FUNCTION_BLOCK FLOOR2_AR (* AR/ADI-Adapter-Wrapper um OSCAT FLOOR2 - bruckt zwischen adapter und OSCAT, ohne dass eine der beiden Basisbibliotheken von der anderen abhaengt *)
  (* Standard: 61499-2; Description: Copyright (c) 2026 Meisterschulen am Ostbahnhof This program and the accompanying materials are made available under the terms of the Eclipse Public License 2.0 which is available at https://www.eclipse.org/legal/epl-2.0/ SPDX-License-Identifier: EPL-2.0 *)
  (* Version 1.0, 2026-09-17, Franz Höpfinger, Meisterschulen am Ostbahnhof, Initial implementation of FLOOR2_AR wrapper FB - E_D_FF_ANY_1 als Aenderungsfilter (EO/ADI_OUT.E1 nur bei tatsaechlicher Wertaenderung), analog CTRL_PI_AR/FT_DERIV_AR in diesem Projekt *)
  PACKAGE OSCAT_adapter::Mathematical;
  (* Documentation:
  FLOOR2_AR
   🇩🇪 Deutsch
   Adapter-Wrapper um OSCAT::Basic::POUs::Mathematical::FLOOR2 (groesste ganze Zahl <= X, DINT-Variante von FLOOR fuer Werte ausserhalb des INT-Bereichs).
   Reine Adapter-Grenze
    - AR_IN (Socket, AR): Eingangssignal (REAL)
   - ADI_OUT (Plug, ADI): Ergebnis (DINT)
    E_D_FF_ANY_1 (Standardbibliothek events-3.0.0) filtert Aenderungen: ADI_OUT.E1 feuert nur, wenn sich das Ergebnis seit dem letzten Aufruf tatsaechlich geaendert hat - gleiches Muster wie bei den bestehenden FT_DERIV_AR/CTRL_PI_AR-Wrappern in diesem Projekt.
   Warum ein eigener Wrapper?
   FLOOR2 ist eine reine OSCAT-Function ohne Adapter-Schnittstelle. adapter soll nicht von OSCAT abhaengen (und umgekehrt) - die Bruecke liegt daher in diesem dritten Bibliotheksprojekt (OSCAT_adapter), das von beiden abhaengt.
   🇬🇧 English
   Adapter wrapper around OSCAT::Basic::POUs::Mathematical::FLOOR2 (largest integer <= X, DINT variant of FLOOR for values outside the INT range).
   Pure adapter boundary
    - AR_IN (socket, AR): input signal (REAL)
   - ADI_OUT (plug, ADI): result (DINT)
    E_D_FF_ANY_1 (standard library events-3.0.0) filters changes: ADI_OUT.E1 only fires when the result actually changed since the last call - same pattern as the existing FT_DERIV_AR/CTRL_PI_AR wrappers in this project.
  *)
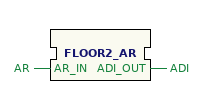
  SOCKETS
    AR_IN : adapter::types::unidirectional::AR; (* Eingangssignal (REAL) *)
  END_SOCKETS
  PLUGS
    ADI_OUT : adapter::types::unidirectional::ADI; (* Groesste ganze Zahl <= X (DINT) *)
  END_PLUGS
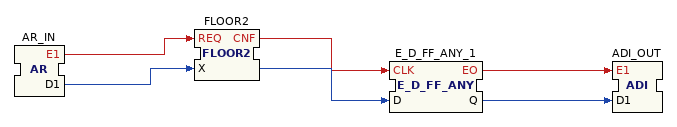
  FBS
    FLOOR2 : OSCAT::Basic::POUs::Mathematical::FLOOR2;
    E_D_FF_ANY_1 : iec61499::events::E_D_FF_ANY;
  END_FBS
  EVENT_CONNECTIONS
    AR_IN.E1 TO FLOOR2.REQ;
    FLOOR2.CNF TO E_D_FF_ANY_1.CLK;
    E_D_FF_ANY_1.EO TO ADI_OUT.E1;
  END_CONNECTIONS
  DATA_CONNECTIONS
    AR_IN.D1 TO FLOOR2.X;
    FLOOR2. TO E_D_FF_ANY_1.D;
    E_D_FF_ANY_1.Q TO ADI_OUT.D1;
  END_CONNECTIONS
END_FUNCTION_BLOCK
